% RSLogix 500 project LVD180611.RSS, saved by version 10.00.00.00 %
PROJECT "LINCEBOT"    % processor: MicroLogix 1400 %

PROGRAM FILES
  LAD 2 "MAIN"  15 rungs  % Main Program Routine %
  LAD 4 "PACKAGER"  10 rungs  % normal %
  LAD 6 "TIMING"  11 rungs  % normal %
  LAD 8 "LOOP TIME"  6 rungs
  LAD 10 "AIR PRESUR"  5 rungs
  LAD 12 "ENABLES"  10 rungs
  LAD 14 "SPEED OUT"  11 rungs
  LAD 70 "OFFSETS"  1 rungs  % normal %
  LAD 80 "HSC BOT"  9 rungs
  LAD 90 "HSC TOP"  9 rungs
  LAD 100 "1 MS STI"  23 rungs  % high speed %
  LAD 102 "SPEED BOT"  6 rungs  % high speed %
  LAD 103 "SPEED TOP"  6 rungs  % high speed %
  LAD 104 "P BOT"  8 rungs  % high speed %
  LAD 105 "P TOP"  8 rungs  % high speed %
  LAD 110 "SHIFT BOT"  5 rungs
  LAD 111 "SHIFT TOP"  5 rungs
  LAD 121 "OPTIC BOT"  23 rungs
  LAD 125 "INS 1"  61 rungs
  LAD 130 "XFER"  6 rungs
  LAD 140 "OPTIC TOP"  37 rungs
  LAD 150 "INS 5"  61 rungs
  LAD 160 "INS 6"  61 rungs
  LAD 170 "PASS BLOW"  3 rungs

DATA FILES
  O0 OUTPUT  11 elements
  I1 INPUT  11 elements
  S2 STATUS  66 elements
  B3 BINARY  14 elements
  T4 TIMER  40 elements
  C5 COUNTER  1 elements
  R6 CONTROL  10 elements
  N7 INTEGER  200 elements
  F8 FLOAT  100 elements
  B9 TOP BS DAT  256 elements
  B10 OLD_COM  1 elements
  B11 BOT BS DAT  256 elements
  B12 HMI_BINARY  22 elements  % general use with hmi to avoid additional reads %
  L13  COUNTS  100 elements
  F14 HMI_FLOAT  100 elements
  N15 HMI_INTS  100 elements
  L16 HMI_LONGS  100 elements
  L23 NEW READ  100 elements
  L24 NEW WRITE  100 elements
  L42   52 elements
  B181 BLANK  128 elements  % used to wipe bs files %
  F182 TEST FLOAT  50 elements
  L183 TEST LONG  50 elements
  N184 TEST INTS  50 elements
  B185 TEST BITS  50 elements
  N186 HMI INTS  50 elements
  L187 HMI LONG  50 elements
  F188 HMI FLOAT  50 elements
  B189 HMI BITS  50 elements
  L190 COUNTS  50 elements
  B191 ERROR BITS  10 elements
  L192 SPD OFFSET  50 elements
  F193 SPD OFFSET  50 elements
  B194 BOT GOOD  128 elements
  B195 TOP GOOD  128 elements
  B196 CTRL BITS  50 elements
  N197 CTRL INTS  50 elements
  B198 TRK BITS  50 elements
  L199 TRK LONG  50 elements
  N200 TRK INTS  50 elements
  L201 INS LONG  50 elements
  B202 INS BITS  50 elements
  N203 INS INTS  50 elements
  L204 CTRL LONG  50 elements
  F205 CTRL FLTS  50 elements

LADDER 2 "MAIN"    % Main Program Routine %
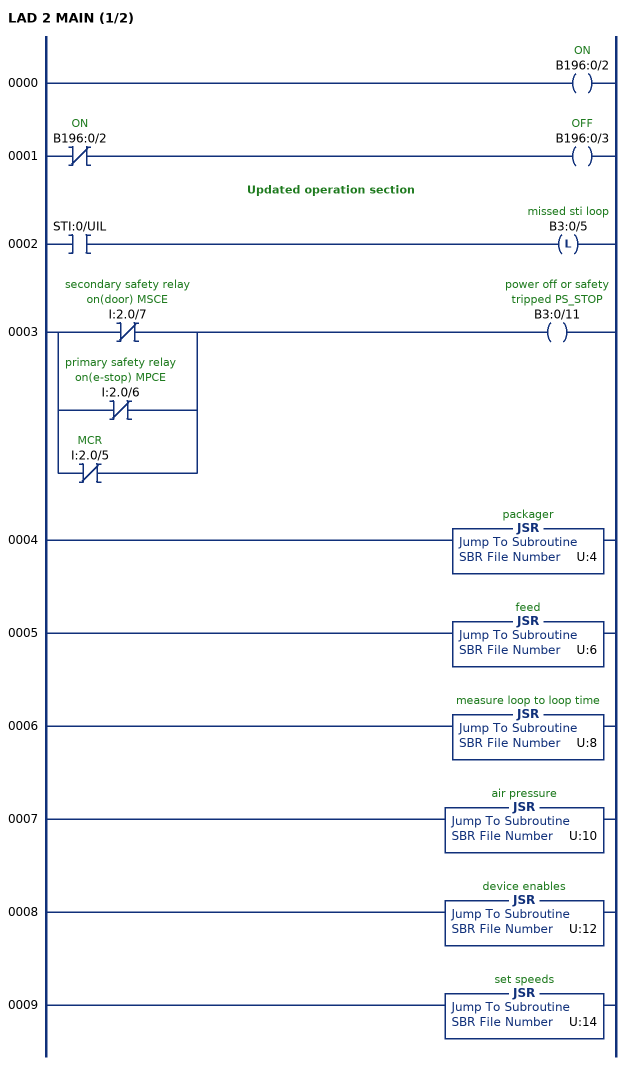
% Rung: 0 %
SOR OTE B196:0/2 EOR
%   B196:0/2  ON %
% Rung: 1 %
SOR XIO B196:0/2 OTE B196:0/3 EOR
%   B196:0/2  ON %
%   B196:0/3  OFF %
% Rung: 2 %
% TITLE: Updated operation section %
SOR XIC STI:0/UIL OTL B3:0/5 EOR
%   B3:0/5  "missed sti loop" %
% Rung: 3 %
SOR BST XIO I:2.0/7 NXB XIO I:2.0/6 NXB XIO I:2.0/5 BND OTE B3:0/11 EOR
%   I:2.0/7  MSCE  "secondary safety relay on(door)" %
%   I:2.0/6  MPCE  "primary safety relay on(e-stop)" %
%   I:2.0/5  MCR %
%   B3:0/11  PS_STOP  "power off or safety tripped" %
% Rung: 4 %
SOR JSR U:4 EOR
%   U:4  "packager" %
% Rung: 5 %
SOR JSR U:6 EOR
%   U:6  "feed" %
% Rung: 6 %
SOR JSR U:8 EOR
%   U:8  "measure loop to loop time" %
% Rung: 7 %
SOR JSR U:10 EOR
%   U:10  "air pressure" %
% Rung: 8 %
SOR JSR U:12 EOR
%   U:12  "device enables" %
% Rung: 9 %
SOR JSR U:14 EOR
%   U:14  "set speeds" %

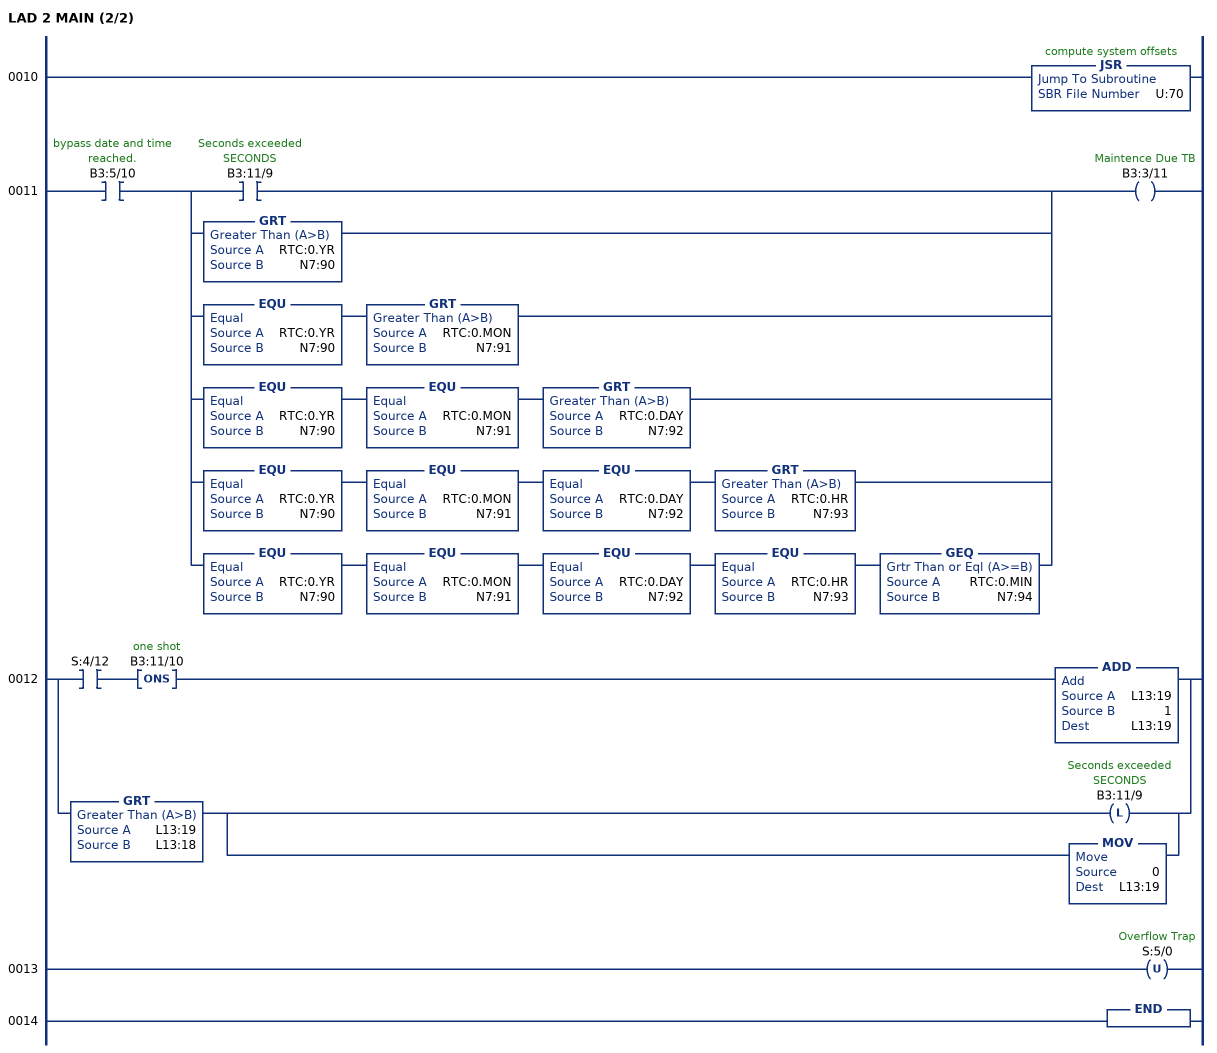
% Rung: 10 %
SOR JSR U:70 EOR
%   U:70  "compute system offsets" %
% Rung: 11 %
SOR XIC B3:5/10 BST XIC B3:11/9 NXB GRT RTC:0.YR N7:90 NXB EQU RTC:0.YR N7:90 GRT RTC:0.MON N7:91 NXB EQU RTC:0.YR N7:90 EQU RTC:0.MON N7:91 GRT RTC:0.DAY N7:92 NXB EQU RTC:0.YR N7:90 EQU RTC:0.MON N7:91 EQU RTC:0.DAY N7:92 GRT RTC:0.HR N7:93 NXB EQU RTC:0.YR N7:90 EQU RTC:0.MON N7:91 EQU RTC:0.DAY N7:92 EQU RTC:0.HR N7:93 GEQ RTC:0.MIN N7:94 BND OTE B3:3/11 EOR
%   B3:5/10  "bypass date and time reached." %
%   B3:11/9  SECONDS  "Seconds exceeded" %
%   N7:90  RTC %
%   B3:3/11  TB  "Maintence Due" %
% Rung: 12 %
SOR BST XIC S:4/12 ONS B3:11/10 ADD L13:19 1 L13:19 NXB GRT L13:19 L13:18 BST OTL B3:11/9 NXB MOV 0 L13:19 BND BND EOR
%   B3:11/10  "one shot" %
%   L13:18  MAX %
%   B3:11/9  SECONDS  "Seconds exceeded" %
% Rung: 13 %
SOR OTU S:5/0 EOR
%   S:5/0  "Overflow Trap" %
% Rung: 14 %
SOR END EOR

LADDER 4 "PACKAGER"    % normal %
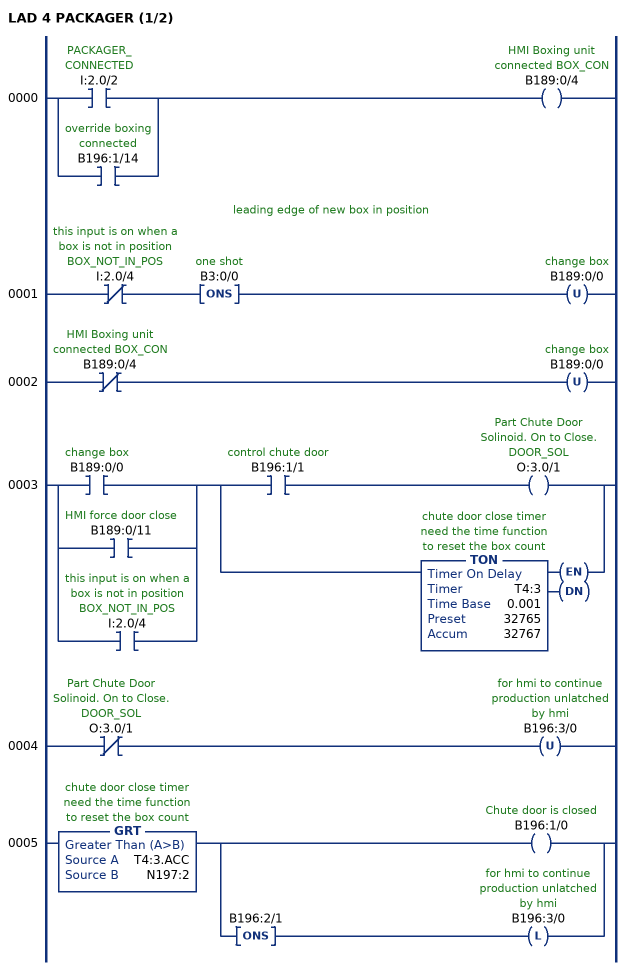
% Rung: 0 %
SOR BST XIC I:2.0/2 NXB XIC B196:1/14 BND OTE B189:0/4 EOR
%   I:2.0/2  PACKAGER_CONNECTED %
%   B196:1/14  "override boxing connected" %
%   B189:0/4  BOX_CON  "HMI Boxing unit connected" %
% Rung: 1 %
% leading edge of new box in position %
SOR XIO I:2.0/4 ONS B3:0/0 OTU B189:0/0 EOR
%   I:2.0/4  BOX_NOT_IN_POS  "this input is on when a box is not in position" %
%   B3:0/0  "one shot" %
%   B189:0/0  "change box" %
% Rung: 2 %
SOR XIO B189:0/4 OTU B189:0/0 EOR
%   B189:0/4  BOX_CON  "HMI Boxing unit connected" %
%   B189:0/0  "change box" %
% Rung: 3 %
SOR BST XIC B189:0/0 NXB XIC B189:0/11 NXB XIC I:2.0/4 BND BST XIC B196:1/1 OTE O:3.0/1 NXB TON T4:3 0.001 32765 32767 BND EOR
%   B189:0/0  "change box" %
%   B189:0/11  "HMI force door close" %
%   I:2.0/4  BOX_NOT_IN_POS  "this input is on when a box is not in position" %
%   B196:1/1  "control chute door" %
%   O:3.0/1  DOOR_SOL  "Part Chute Door Solinoid. On to Close." %
%   T4:3  "chute door close timer need the time function to reset the box count" %
% Rung: 4 %
SOR XIO O:3.0/1 OTU B196:3/0 EOR
%   O:3.0/1  DOOR_SOL  "Part Chute Door Solinoid. On to Close." %
%   B196:3/0  "for hmi to continue production unlatched by hmi" %
% Rung: 5 %
SOR GRT T4:3.ACC N197:2 BST OTE B196:1/0 NXB ONS B196:2/1 OTL B196:3/0 BND EOR
%   T4:3  "chute door close timer need the time function to reset the box count" %
%   N197:2  "time for chute door to close" %
%   B196:1/0  "Chute door is closed" %
%   B196:3/0  "for hmi to continue production unlatched by hmi" %

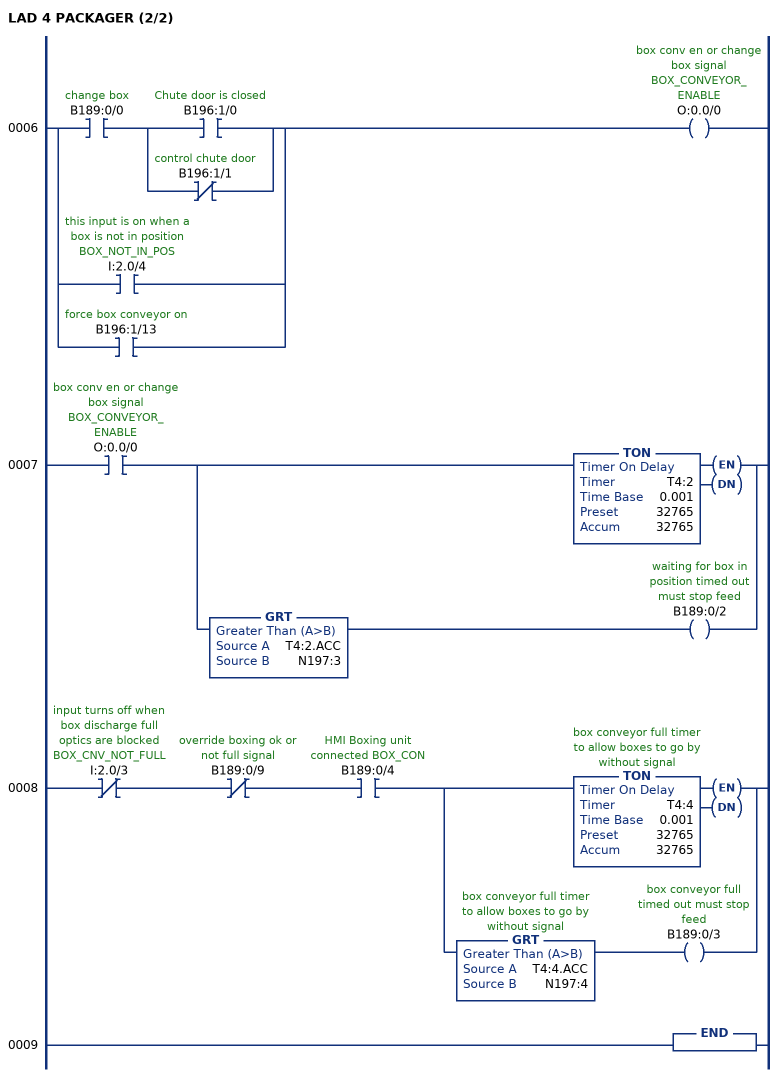
% Rung: 6 %
SOR BST XIC B189:0/0 BST XIC B196:1/0 NXB XIO B196:1/1 BND NXB XIC I:2.0/4 NXB XIC B196:1/13 BND OTE O:0.0/0 EOR
%   B189:0/0  "change box" %
%   B196:1/0  "Chute door is closed" %
%   B196:1/1  "control chute door" %
%   I:2.0/4  BOX_NOT_IN_POS  "this input is on when a box is not in position" %
%   B196:1/13  "force box conveyor on" %
%   O:0.0/0  BOX_CONVEYOR_ENABLE  "box conv en or change box signal" %
% Rung: 7 %
SOR XIC O:0.0/0 BST TON T4:2 0.001 32765 32765 NXB GRT T4:2.ACC N197:3 OTE B189:0/2 BND EOR
%   O:0.0/0  BOX_CONVEYOR_ENABLE  "box conv en or change box signal" %
%   N197:3  "FeedWheel Speed Output Setting" %
%   B189:0/2  "waiting for box in position timed out must stop feed" %
% Rung: 8 %
SOR XIO I:2.0/3 XIO B189:0/9 XIC B189:0/4 BST TON T4:4 0.001 32765 32765 NXB GRT T4:4.ACC N197:4 OTE B189:0/3 BND EOR
%   I:2.0/3  BOX_CNV_NOT_FULL  "input turns off when box discharge full optics are blocked" %
%   B189:0/9  "override boxing ok or not full signal" %
%   B189:0/4  BOX_CON  "HMI Boxing unit connected" %
%   T4:4  "box conveyor full timer to allow boxes to go by without signal" %
%   N197:4  "boxing convery full time out time (ms)" %
%   B189:0/3  "box conveyor full timed out must stop feed" %
% Rung: 9 %
SOR END EOR

LADDER 6 "TIMING"    % normal %
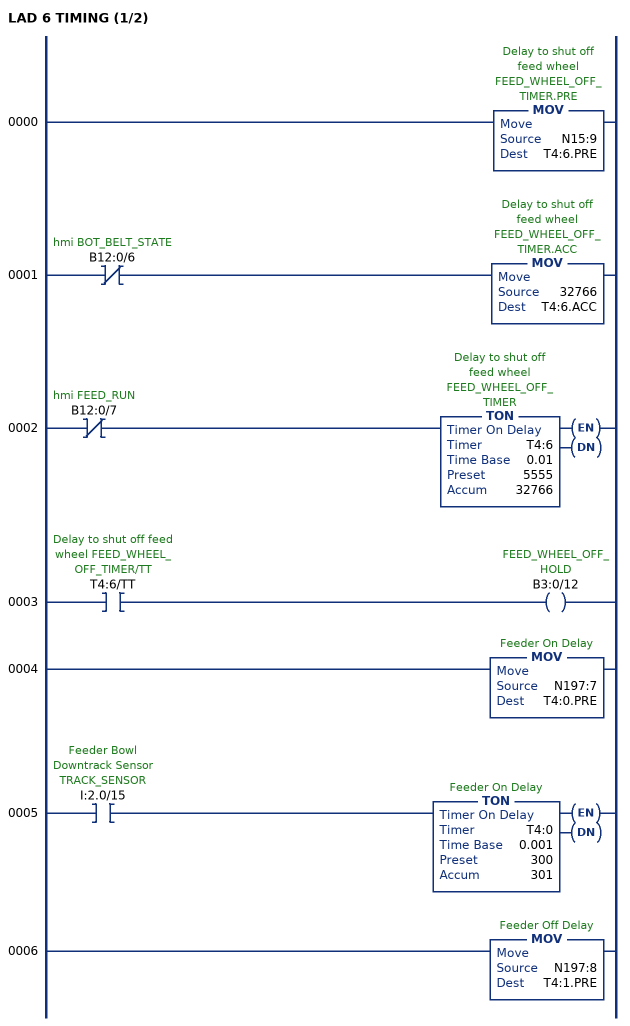
% Rung: 0 %
SOR MOV N15:9 T4:6.PRE EOR
%   N15:9  FEED_WHEEL_STOP_TIME %
%   T4:6  FEED_WHEEL_OFF_TIMER  "Delay to shut off feed wheel" %
% Rung: 1 %
SOR XIO B12:0/6 MOV 32766 T4:6.ACC EOR
%   B12:0/6  BOT_BELT_STATE  "hmi" %
%   T4:6  FEED_WHEEL_OFF_TIMER  "Delay to shut off feed wheel" %
% Rung: 2 %
SOR XIO B12:0/7 TON T4:6 0.01 5555 32766 EOR
%   B12:0/7  FEED_RUN  "hmi" %
%   T4:6  FEED_WHEEL_OFF_TIMER  "Delay to shut off feed wheel" %
% Rung: 3 %
SOR XIC T4:6/TT OTE B3:0/12 EOR
%   T4:6  FEED_WHEEL_OFF_TIMER  "Delay to shut off feed wheel" %
%   B3:0/12  FEED_WHEEL_OFF_HOLD %
% Rung: 4 %
SOR MOV N197:7 T4:0.PRE EOR
%   N197:7  "down track on delay" %
%   T4:0  "Feeder On Delay" %
% Rung: 5 %
SOR XIC I:2.0/15 TON T4:0 0.001 300 301 EOR
%   I:2.0/15  TRACK_SENSOR  "Feeder Bowl Downtrack Sensor" %
%   T4:0  "Feeder On Delay" %
% Rung: 6 %
SOR MOV N197:8 T4:1.PRE EOR
%   N197:8  "down track off delay" %
%   T4:1  "Feeder Off Delay" %

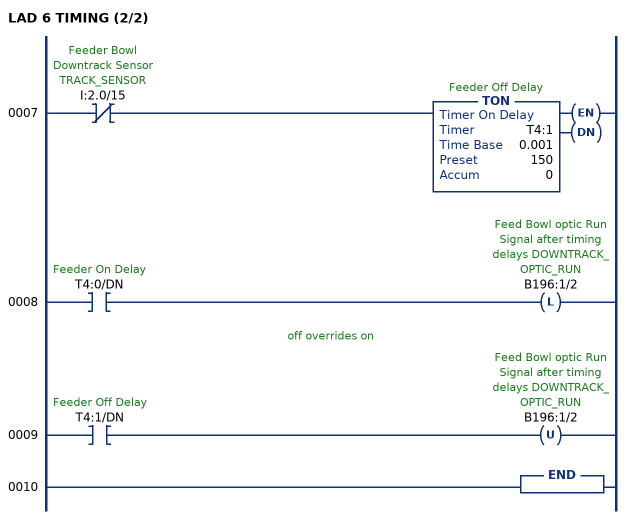
% Rung: 7 %
SOR XIO I:2.0/15 TON T4:1 0.001 150 0 EOR
%   I:2.0/15  TRACK_SENSOR  "Feeder Bowl Downtrack Sensor" %
%   T4:1  "Feeder Off Delay" %
% Rung: 8 %
SOR XIC T4:0/DN OTL B196:1/2 EOR
%   T4:0  "Feeder On Delay" %
%   B196:1/2  DOWNTRACK_OPTIC_RUN  "Feed Bowl optic Run Signal after timing delays" %
% Rung: 9 %
% off overrides on %
SOR XIC T4:1/DN OTU B196:1/2 EOR
%   T4:1  "Feeder Off Delay" %
%   B196:1/2  DOWNTRACK_OPTIC_RUN  "Feed Bowl optic Run Signal after timing delays" %
% Rung: 10 %
SOR END EOR

LADDER 8 "LOOP TIME"
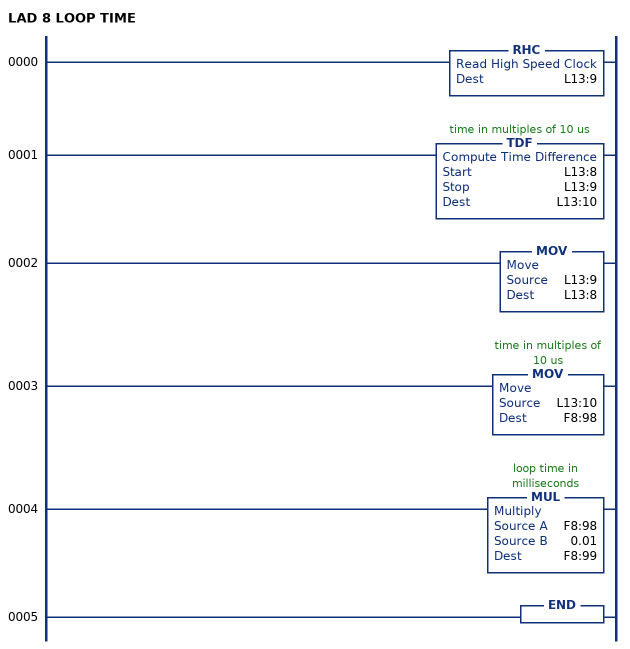
% Rung: 0 %
SOR RHC L13:9 EOR
% Rung: 1 %
SOR TDF L13:8 L13:9 L13:10 EOR
%   L13:10  "time in multiples of 10 us" %
% Rung: 2 %
SOR MOV L13:9 L13:8 EOR
% Rung: 3 %
SOR MOV L13:10 F8:98 EOR
%   L13:10  "time in multiples of 10 us" %
%   F8:98  "time in multiples of 10 us" %
% Rung: 4 %
SOR MUL F8:98 0.01 F8:99 EOR
%   F8:98  "time in multiples of 10 us" %
%   F8:99  "loop time in milliseconds" %
% Rung: 5 %
SOR END EOR

LADDER 10 "AIR PRESUR"
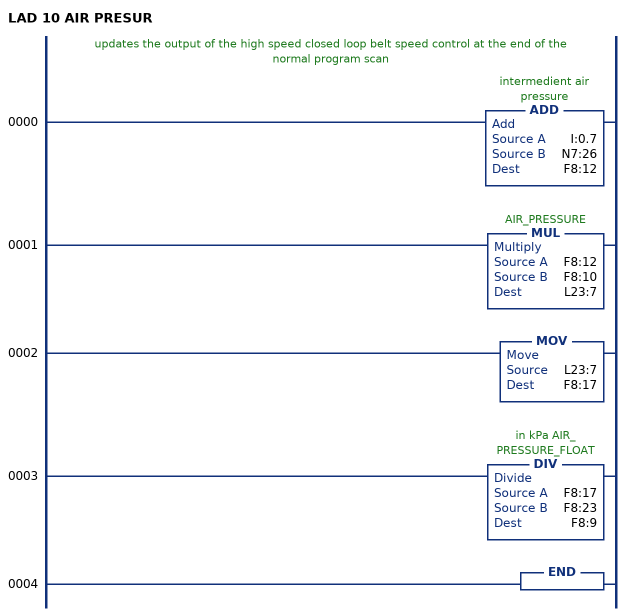
% Rung: 0 %
% updates the output of the high speed closed loop belt speed control at the end of the normal program scan %
SOR ADD I:0.7 N7:26 F8:12 EOR
%   I:0.7  "Air Presure Sensor Input Signal" %
%   N7:26  MAIN_AIR_OFFSET  "Main Air Offset old machine -398 new machine 0" %
%   F8:12  "intermedient air pressure" %
% Rung: 1 %
SOR MUL F8:12 F8:10 L23:7 EOR
%   F8:12  "intermedient air pressure" %
%   F8:10  AIR_MULTIPLIER_BAR  "Air Multiplier (BAR)" %
%   L23:7  AIR_PRESSURE %
% Rung: 2 %
SOR MOV L23:7 F8:17 EOR
%   L23:7  AIR_PRESSURE %
% Rung: 3 %
SOR DIV F8:17 F8:23 F8:9 EOR
%   F8:9  AIR_PRESSURE_FLOAT  "in kPa" %
% Rung: 4 %
SOR END EOR

LADDER 12 "ENABLES"
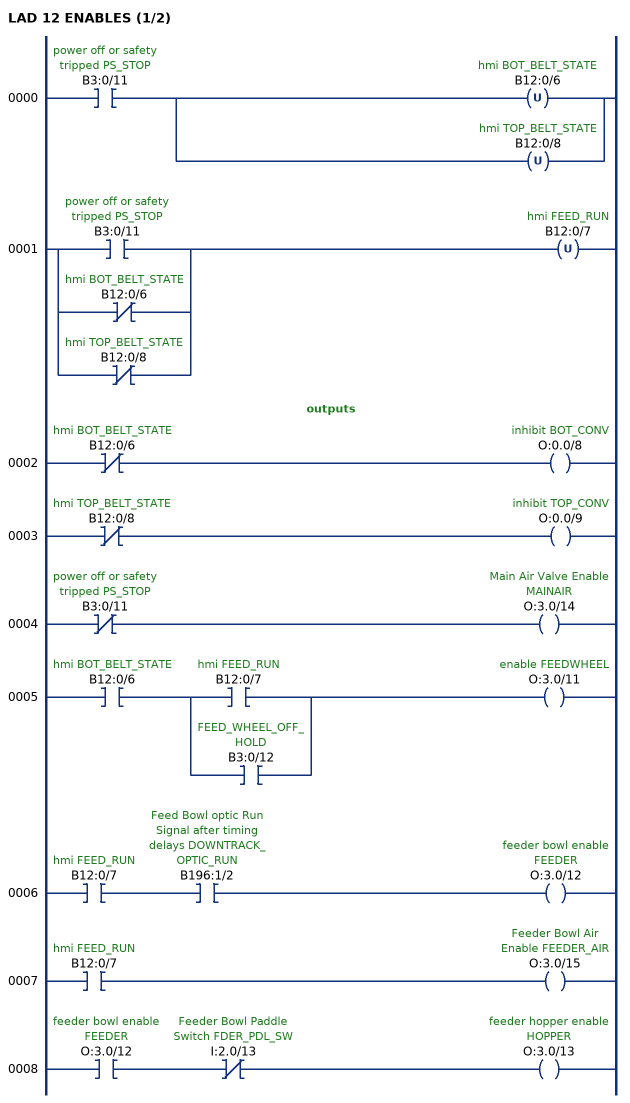
% Rung: 0 %
SOR XIC B3:0/11 BST OTU B12:0/6 NXB OTU B12:0/8 BND EOR
%   B3:0/11  PS_STOP  "power off or safety tripped" %
%   B12:0/6  BOT_BELT_STATE  "hmi" %
%   B12:0/8  TOP_BELT_STATE  "hmi" %
% Rung: 1 %
SOR BST XIC B3:0/11 NXB XIO B12:0/6 NXB XIO B12:0/8 BND OTU B12:0/7 EOR
%   B3:0/11  PS_STOP  "power off or safety tripped" %
%   B12:0/6  BOT_BELT_STATE  "hmi" %
%   B12:0/8  TOP_BELT_STATE  "hmi" %
%   B12:0/7  FEED_RUN  "hmi" %
% Rung: 2 %
% TITLE: outputs %
SOR XIO B12:0/6 OTE O:0.0/8 EOR
%   B12:0/6  BOT_BELT_STATE  "hmi" %
%   O:0.0/8  BOT_CONV  "inhibit" %
% Rung: 3 %
SOR XIO B12:0/8 OTE O:0.0/9 EOR
%   B12:0/8  TOP_BELT_STATE  "hmi" %
%   O:0.0/9  TOP_CONV  "inhibit" %
% Rung: 4 %
SOR XIO B3:0/11 OTE O:3.0/14 EOR
%   B3:0/11  PS_STOP  "power off or safety tripped" %
%   O:3.0/14  MAINAIR  "Main Air Valve Enable" %
% Rung: 5 %
SOR XIC B12:0/6 BST XIC B12:0/7 NXB XIC B3:0/12 BND OTE O:3.0/11 EOR
%   B12:0/6  BOT_BELT_STATE  "hmi" %
%   B12:0/7  FEED_RUN  "hmi" %
%   B3:0/12  FEED_WHEEL_OFF_HOLD %
%   O:3.0/11  FEEDWHEEL  "enable" %
% Rung: 6 %
SOR XIC B12:0/7 XIC B196:1/2 OTE O:3.0/12 EOR
%   B12:0/7  FEED_RUN  "hmi" %
%   B196:1/2  DOWNTRACK_OPTIC_RUN  "Feed Bowl optic Run Signal after timing delays" %
%   O:3.0/12  FEEDER  "feeder bowl enable" %
% Rung: 7 %
SOR XIC B12:0/7 OTE O:3.0/15 EOR
%   B12:0/7  FEED_RUN  "hmi" %
%   O:3.0/15  FEEDER_AIR  "Feeder Bowl Air Enable" %
% Rung: 8 %
SOR XIC O:3.0/12 XIO I:2.0/13 OTE O:3.0/13 EOR
%   O:3.0/12  FEEDER  "feeder bowl enable" %
%   I:2.0/13  FDER_PDL_SW  "Feeder Bowl Paddle Switch" %
%   O:3.0/13  HOPPER  "feeder hopper enable" %

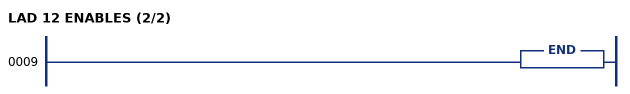
% Rung: 9 %
SOR END EOR

LADDER 14 "SPEED OUT"
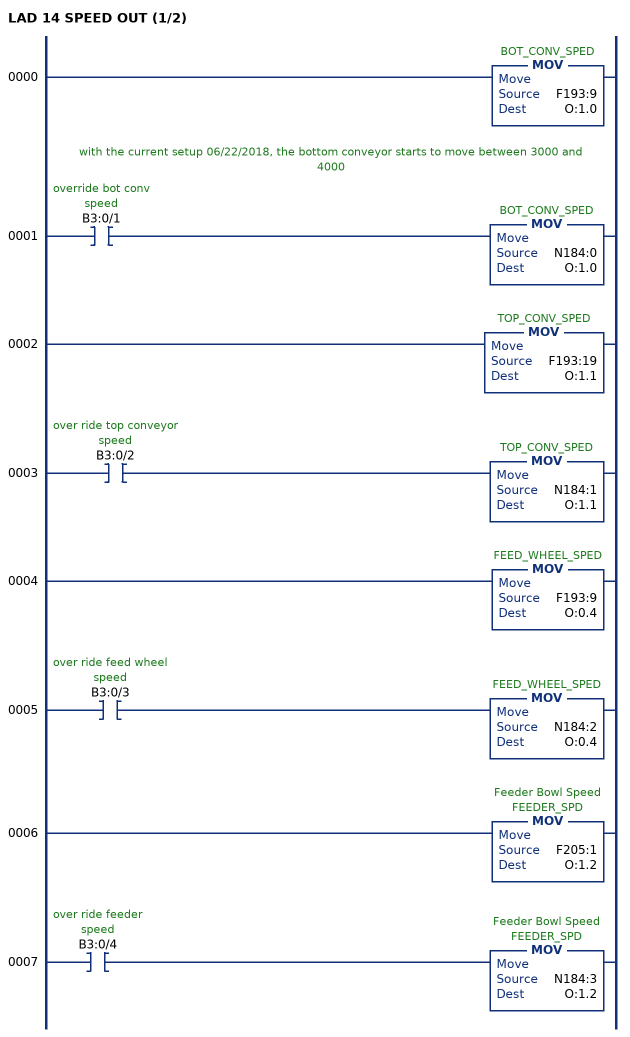
% Rung: 0 %
SOR MOV F193:9 O:1.0 EOR
%   F193:9  SCALED_BOT_VALUE %
%   O:1.0  BOT_CONV_SPED %
% Rung: 1 %
% with the current setup 06/22/2018, the bottom conveyor starts to move between 3000 and 4000 %
SOR XIC B3:0/1 MOV N184:0 O:1.0 EOR
%   B3:0/1  "override bot conv speed" %
%   O:1.0  BOT_CONV_SPED %
% Rung: 2 %
SOR MOV F193:19 O:1.1 EOR
%   F193:19  SCALED_TOP_VALUE %
%   O:1.1  TOP_CONV_SPED %
% Rung: 3 %
SOR XIC B3:0/2 MOV N184:1 O:1.1 EOR
%   B3:0/2  "over ride top conveyor speed" %
%   O:1.1  TOP_CONV_SPED %
% Rung: 4 %
SOR MOV F193:9 O:0.4 EOR
%   F193:9  SCALED_BOT_VALUE %
%   O:0.4  FEED_WHEEL_SPED %
% Rung: 5 %
SOR XIC B3:0/3 MOV N184:2 O:0.4 EOR
%   B3:0/3  "over ride feed wheel speed" %
%   O:0.4  FEED_WHEEL_SPED %
% Rung: 6 %
SOR MOV F205:1 O:1.2 EOR
%   F205:1  "feed bowl" %
%   O:1.2  FEEDER_SPD  "Feeder Bowl Speed" %
% Rung: 7 %
SOR XIC B3:0/4 MOV N184:3 O:1.2 EOR
%   B3:0/4  "over ride feeder speed" %
%   O:1.2  FEEDER_SPD  "Feeder Bowl Speed" %

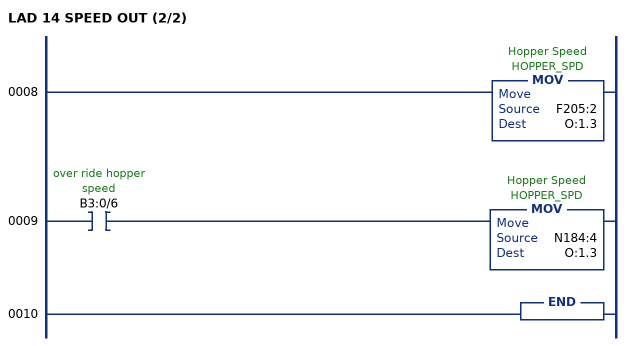
% Rung: 8 %
SOR MOV F205:2 O:1.3 EOR
%   F205:2  "hopper" %
%   O:1.3  HOPPER_SPD  "Hopper Speed" %
% Rung: 9 %
SOR XIC B3:0/6 MOV N184:4 O:1.3 EOR
%   B3:0/6  "over ride hopper speed" %
%   O:1.3  HOPPER_SPD  "Hopper Speed" %
% Rung: 10 %
SOR END EOR

LADDER 80 "HSC BOT"
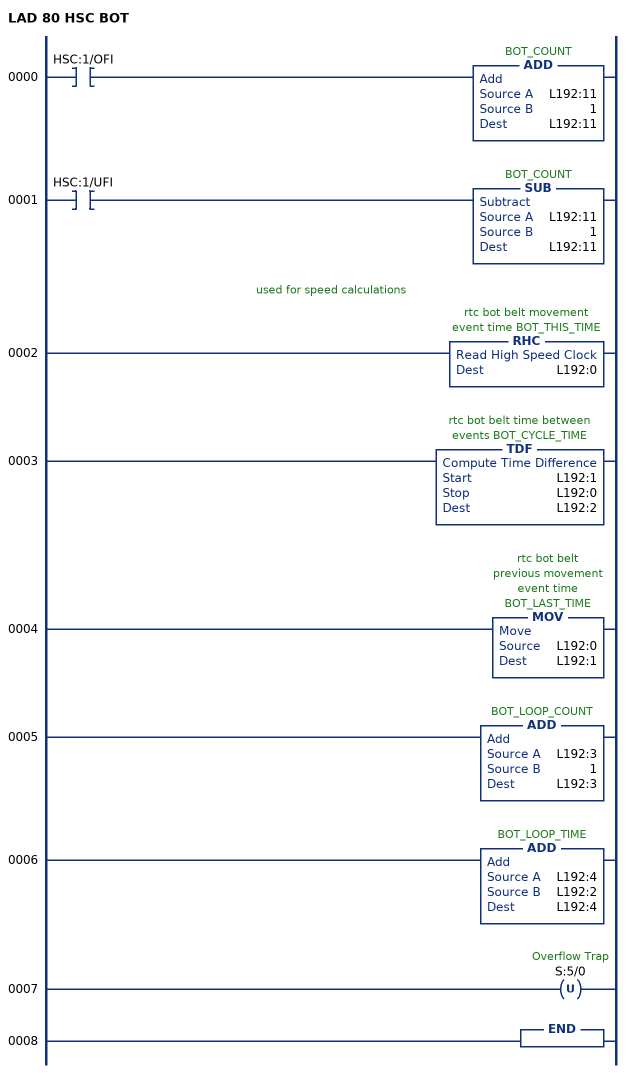
% Rung: 0 %
SOR XIC HSC:1/OFI ADD L192:11 1 L192:11 EOR
%   L192:11  BOT_COUNT %
% Rung: 1 %
SOR XIC HSC:1/UFI SUB L192:11 1 L192:11 EOR
%   L192:11  BOT_COUNT %
% Rung: 2 %
% used for speed calculations %
SOR RHC L192:0 EOR
%   L192:0  BOT_THIS_TIME  "rtc bot belt movement event time" %
% Rung: 3 %
SOR TDF L192:1 L192:0 L192:2 EOR
%   L192:1  BOT_LAST_TIME  "rtc bot belt previous movement event time" %
%   L192:0  BOT_THIS_TIME  "rtc bot belt movement event time" %
%   L192:2  BOT_CYCLE_TIME  "rtc bot belt time between events" %
% Rung: 4 %
SOR MOV L192:0 L192:1 EOR
%   L192:0  BOT_THIS_TIME  "rtc bot belt movement event time" %
%   L192:1  BOT_LAST_TIME  "rtc bot belt previous movement event time" %
% Rung: 5 %
SOR ADD L192:3 1 L192:3 EOR
%   L192:3  BOT_LOOP_COUNT %
% Rung: 6 %
SOR ADD L192:4 L192:2 L192:4 EOR
%   L192:4  BOT_LOOP_TIME %
%   L192:2  BOT_CYCLE_TIME  "rtc bot belt time between events" %
% Rung: 7 %
SOR OTU S:5/0 EOR
%   S:5/0  "Overflow Trap" %
% Rung: 8 %
SOR END EOR

LADDER 90 "HSC TOP"
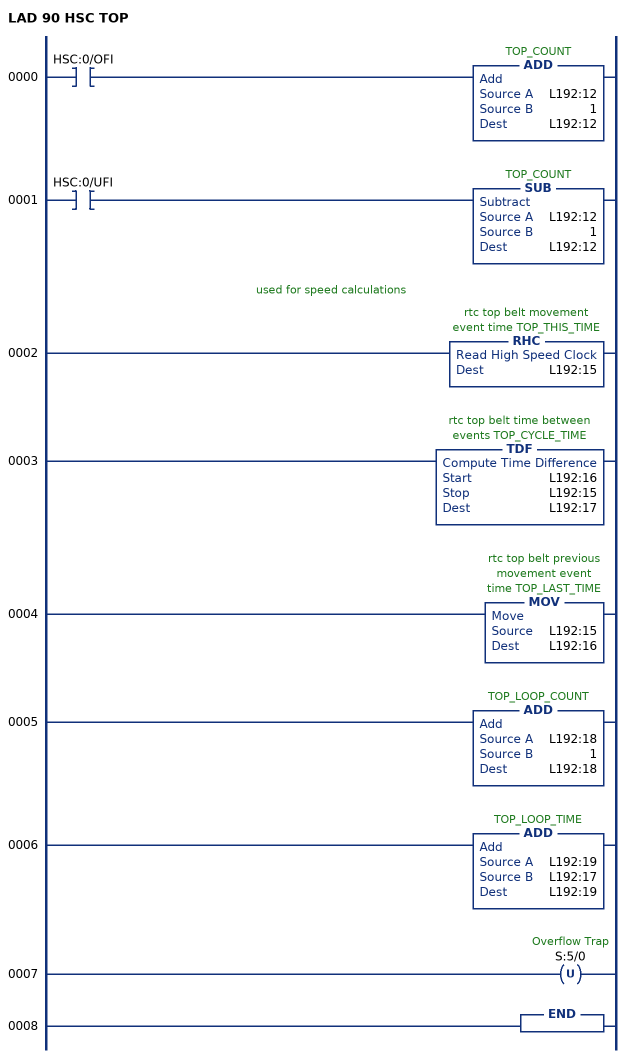
% Rung: 0 %
SOR XIC HSC:0/OFI ADD L192:12 1 L192:12 EOR
%   L192:12  TOP_COUNT %
% Rung: 1 %
SOR XIC HSC:0/UFI SUB L192:12 1 L192:12 EOR
%   L192:12  TOP_COUNT %
% Rung: 2 %
% used for speed calculations %
SOR RHC L192:15 EOR
%   L192:15  TOP_THIS_TIME  "rtc top belt movement event time" %
% Rung: 3 %
SOR TDF L192:16 L192:15 L192:17 EOR
%   L192:16  TOP_LAST_TIME  "rtc top belt previous movement event time" %
%   L192:15  TOP_THIS_TIME  "rtc top belt movement event time" %
%   L192:17  TOP_CYCLE_TIME  "rtc top belt time between events" %
% Rung: 4 %
SOR MOV L192:15 L192:16 EOR
%   L192:15  TOP_THIS_TIME  "rtc top belt movement event time" %
%   L192:16  TOP_LAST_TIME  "rtc top belt previous movement event time" %
% Rung: 5 %
SOR ADD L192:18 1 L192:18 EOR
%   L192:18  TOP_LOOP_COUNT %
% Rung: 6 %
SOR ADD L192:19 L192:17 L192:19 EOR
%   L192:19  TOP_LOOP_TIME %
%   L192:17  TOP_CYCLE_TIME  "rtc top belt time between events" %
% Rung: 7 %
SOR OTU S:5/0 EOR
%   S:5/0  "Overflow Trap" %
% Rung: 8 %
SOR END EOR

LADDER 100 "1 MS STI"    % high speed %
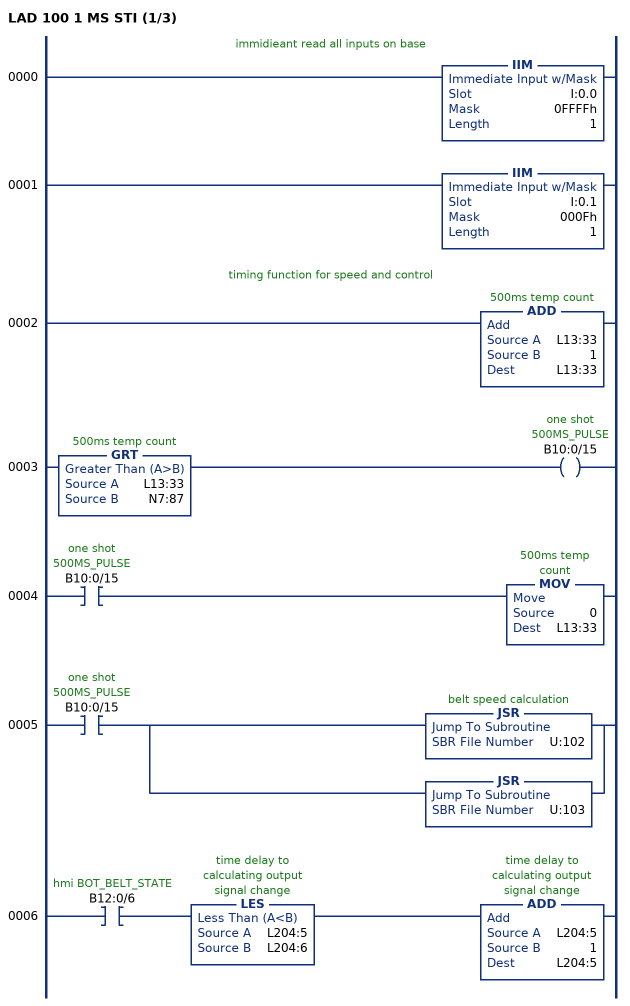
% Rung: 0 %
% immidieant read all inputs on base %
SOR IIM I:0.0 0FFFFh 1 EOR
% Rung: 1 %
SOR IIM I:0.1 000Fh 1 EOR
% Rung: 2 %
% timing function for speed and control %
SOR ADD L13:33 1 L13:33 EOR
%   L13:33  "500ms temp count" %
% Rung: 3 %
SOR GRT L13:33 N7:87 OTE B10:0/15 EOR
%   L13:33  "500ms temp count" %
%   B10:0/15  500MS_PULSE  "one shot" %
% Rung: 4 %
SOR XIC B10:0/15 MOV 0 L13:33 EOR
%   B10:0/15  500MS_PULSE  "one shot" %
%   L13:33  "500ms temp count" %
% Rung: 5 %
SOR XIC B10:0/15 BST JSR U:102 NXB JSR U:103 BND EOR
%   B10:0/15  500MS_PULSE  "one shot" %
%   U:102  "belt speed calculation" %
% Rung: 6 %
SOR XIC B12:0/6 LES L204:5 L204:6 ADD L204:5 1 L204:5 EOR
%   B12:0/6  BOT_BELT_STATE  "hmi" %
%   L204:5  "time delay to calculating output signal change" %
%   L204:6  "belt start delay time" %

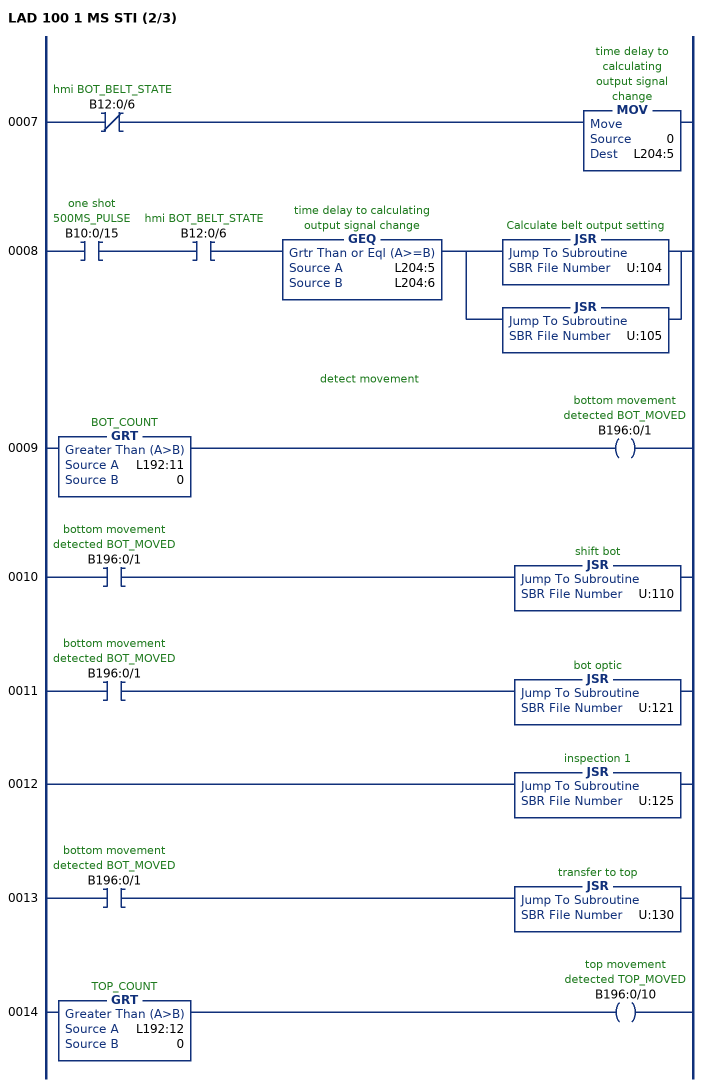
% Rung: 7 %
SOR XIO B12:0/6 MOV 0 L204:5 EOR
%   B12:0/6  BOT_BELT_STATE  "hmi" %
%   L204:5  "time delay to calculating output signal change" %
% Rung: 8 %
SOR XIC B10:0/15 XIC B12:0/6 GEQ L204:5 L204:6 BST JSR U:104 NXB JSR U:105 BND EOR
%   B10:0/15  500MS_PULSE  "one shot" %
%   B12:0/6  BOT_BELT_STATE  "hmi" %
%   L204:5  "time delay to calculating output signal change" %
%   L204:6  "belt start delay time" %
%   U:104  "Calculate belt output setting" %
% Rung: 9 %
% detect movement %
SOR GRT L192:11 0 OTE B196:0/1 EOR
%   L192:11  BOT_COUNT %
%   B196:0/1  BOT_MOVED  "bottom movement detected" %
% Rung: 10 %
SOR XIC B196:0/1 JSR U:110 EOR
%   B196:0/1  BOT_MOVED  "bottom movement detected" %
%   U:110  "shift bot" %
% Rung: 11 %
SOR XIC B196:0/1 JSR U:121 EOR
%   B196:0/1  BOT_MOVED  "bottom movement detected" %
%   U:121  "bot optic" %
% Rung: 12 %
SOR JSR U:125 EOR
%   U:125  "inspection 1" %
% Rung: 13 %
SOR XIC B196:0/1 JSR U:130 EOR
%   B196:0/1  BOT_MOVED  "bottom movement detected" %
%   U:130  "transfer to top" %
% Rung: 14 %
SOR GRT L192:12 0 OTE B196:0/10 EOR
%   L192:12  TOP_COUNT %
%   B196:0/10  TOP_MOVED  "top movement detected" %

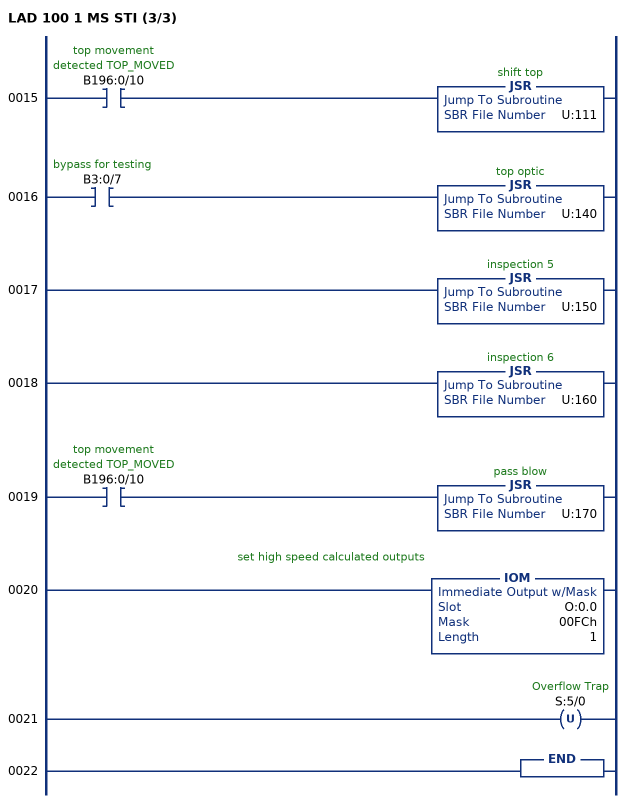
% Rung: 15 %
SOR XIC B196:0/10 JSR U:111 EOR
%   B196:0/10  TOP_MOVED  "top movement detected" %
%   U:111  "shift top" %
% Rung: 16 %
SOR XIC B3:0/7 JSR U:140 EOR
%   B3:0/7  "bypass for testing" %
%   U:140  "top optic" %
% Rung: 17 %
SOR JSR U:150 EOR
%   U:150  "inspection 5" %
% Rung: 18 %
SOR JSR U:160 EOR
%   U:160  "inspection 6" %
% Rung: 19 %
SOR XIC B196:0/10 JSR U:170 EOR
%   B196:0/10  TOP_MOVED  "top movement detected" %
%   U:170  "pass blow" %
% Rung: 20 %
% set high speed calculated outputs %
SOR IOM O:0.0 00FCh 1 EOR
% Rung: 21 %
SOR OTU S:5/0 EOR
%   S:5/0  "Overflow Trap" %
% Rung: 22 %
SOR END EOR

LADDER 102 "SPEED BOT"    % high speed %
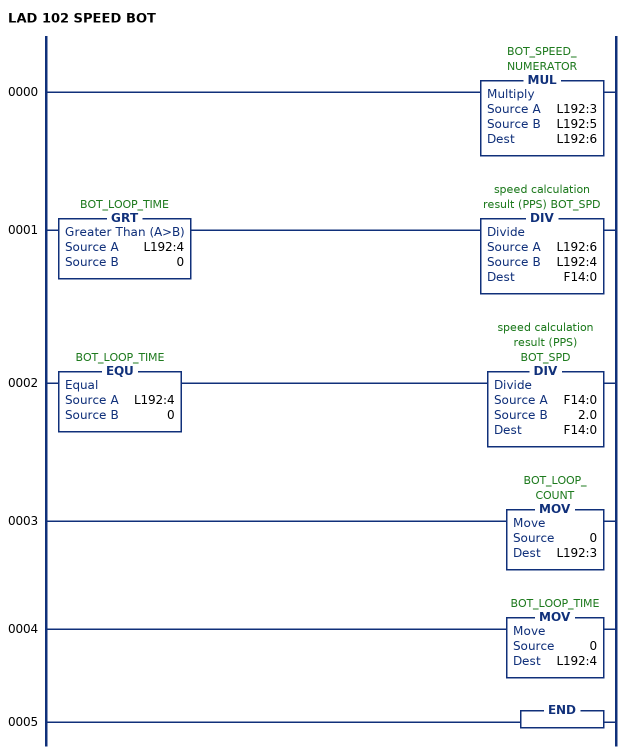
% Rung: 0 %
SOR MUL L192:3 L192:5 L192:6 EOR
%   L192:3  BOT_LOOP_COUNT %
%   L192:5  TKS_PER_SECOND %
%   L192:6  BOT_SPEED_NUMERATOR %
% Rung: 1 %
SOR GRT L192:4 0 DIV L192:6 L192:4 F14:0 EOR
%   L192:4  BOT_LOOP_TIME %
%   L192:6  BOT_SPEED_NUMERATOR %
%   F14:0  BOT_SPD  "speed calculation result (PPS)" %
% Rung: 2 %
SOR EQU L192:4 0 DIV F14:0 2.0 F14:0 EOR
%   L192:4  BOT_LOOP_TIME %
%   F14:0  BOT_SPD  "speed calculation result (PPS)" %
% Rung: 3 %
SOR MOV 0 L192:3 EOR
%   L192:3  BOT_LOOP_COUNT %
% Rung: 4 %
SOR MOV 0 L192:4 EOR
%   L192:4  BOT_LOOP_TIME %
% Rung: 5 %
SOR END EOR

LADDER 103 "SPEED TOP"    % high speed %
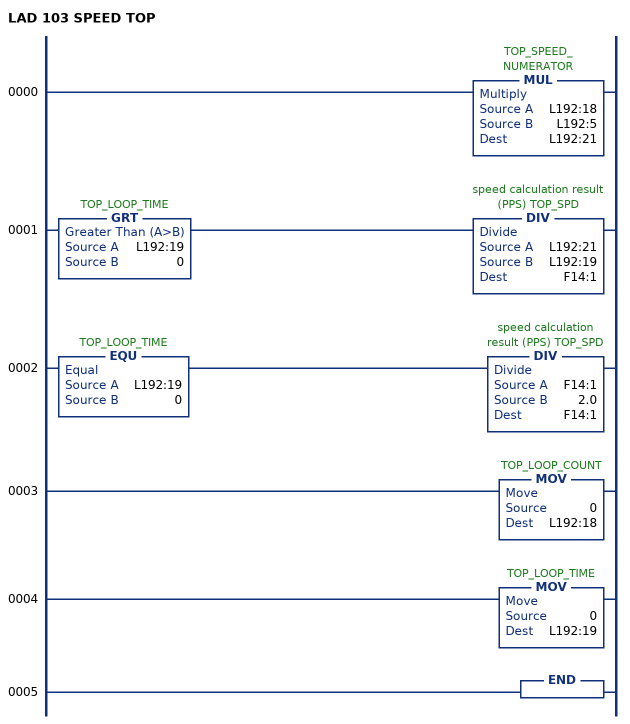
% Rung: 0 %
SOR MUL L192:18 L192:5 L192:21 EOR
%   L192:18  TOP_LOOP_COUNT %
%   L192:5  TKS_PER_SECOND %
%   L192:21  TOP_SPEED_NUMERATOR %
% Rung: 1 %
SOR GRT L192:19 0 DIV L192:21 L192:19 F14:1 EOR
%   L192:19  TOP_LOOP_TIME %
%   L192:21  TOP_SPEED_NUMERATOR %
%   F14:1  TOP_SPD  "speed calculation result (PPS)" %
% Rung: 2 %
SOR EQU L192:19 0 DIV F14:1 2.0 F14:1 EOR
%   L192:19  TOP_LOOP_TIME %
%   F14:1  TOP_SPD  "speed calculation result (PPS)" %
% Rung: 3 %
SOR MOV 0 L192:18 EOR
%   L192:18  TOP_LOOP_COUNT %
% Rung: 4 %
SOR MOV 0 L192:19 EOR
%   L192:19  TOP_LOOP_TIME %
% Rung: 5 %
SOR END EOR

LADDER 104 "P BOT"    % high speed %
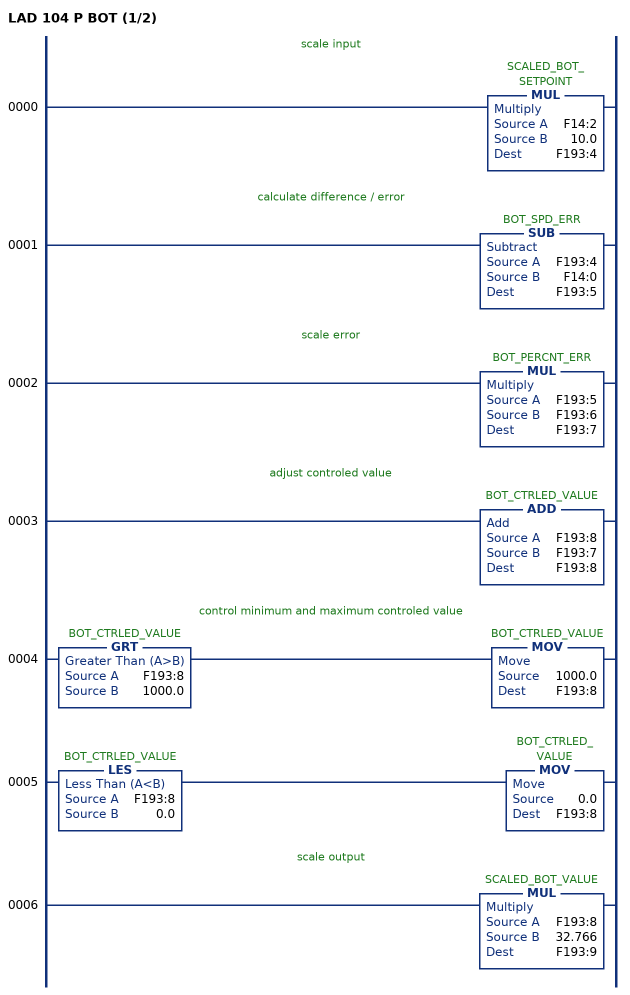
% Rung: 0 %
% scale input %
SOR MUL F14:2 10.0 F193:4 EOR
%   F14:2  BOT_SPD_SETPOINT %
%   F193:4  SCALED_BOT_SETPOINT %
% Rung: 1 %
% calculate difference / error %
SOR SUB F193:4 F14:0 F193:5 EOR
%   F193:4  SCALED_BOT_SETPOINT %
%   F14:0  BOT_SPD  "speed calculation result (PPS)" %
%   F193:5  BOT_SPD_ERR %
% Rung: 2 %
% scale error %
SOR MUL F193:5 F193:6 F193:7 EOR
%   F193:5  BOT_SPD_ERR %
%   F193:6  BOT_FDBK_RATIO %
%   F193:7  BOT_PERCNT_ERR %
% Rung: 3 %
% adjust controled value %
SOR ADD F193:8 F193:7 F193:8 EOR
%   F193:8  BOT_CTRLED_VALUE %
%   F193:7  BOT_PERCNT_ERR %
% Rung: 4 %
% control minimum and maximum controled value %
SOR GRT F193:8 1000.0 MOV 1000.0 F193:8 EOR
%   F193:8  BOT_CTRLED_VALUE %
% Rung: 5 %
SOR LES F193:8 0.0 MOV 0.0 F193:8 EOR
%   F193:8  BOT_CTRLED_VALUE %
% Rung: 6 %
% scale output %
SOR MUL F193:8 32.766 F193:9 EOR
%   F193:8  BOT_CTRLED_VALUE %
%   F193:9  SCALED_BOT_VALUE %

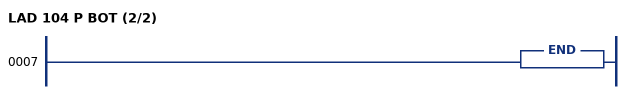
% Rung: 7 %
SOR END EOR

LADDER 105 "P TOP"    % high speed %
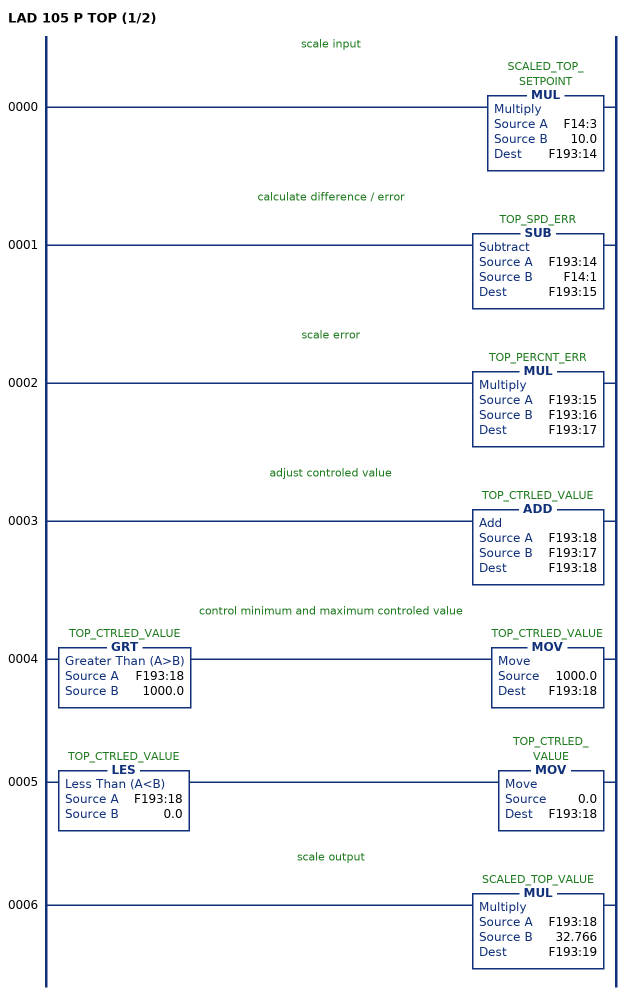
% Rung: 0 %
% scale input %
SOR MUL F14:3 10.0 F193:14 EOR
%   F14:3  TOP_SPD_SETPOINT %
%   F193:14  SCALED_TOP_SETPOINT %
% Rung: 1 %
% calculate difference / error %
SOR SUB F193:14 F14:1 F193:15 EOR
%   F193:14  SCALED_TOP_SETPOINT %
%   F14:1  TOP_SPD  "speed calculation result (PPS)" %
%   F193:15  TOP_SPD_ERR %
% Rung: 2 %
% scale error %
SOR MUL F193:15 F193:16 F193:17 EOR
%   F193:15  TOP_SPD_ERR %
%   F193:16  TOP_FDBK_RATIO %
%   F193:17  TOP_PERCNT_ERR %
% Rung: 3 %
% adjust controled value %
SOR ADD F193:18 F193:17 F193:18 EOR
%   F193:18  TOP_CTRLED_VALUE %
%   F193:17  TOP_PERCNT_ERR %
% Rung: 4 %
% control minimum and maximum controled value %
SOR GRT F193:18 1000.0 MOV 1000.0 F193:18 EOR
%   F193:18  TOP_CTRLED_VALUE %
% Rung: 5 %
SOR LES F193:18 0.0 MOV 0.0 F193:18 EOR
%   F193:18  TOP_CTRLED_VALUE %
% Rung: 6 %
% scale output %
SOR MUL F193:18 32.766 F193:19 EOR
%   F193:18  TOP_CTRLED_VALUE %
%   F193:19  SCALED_TOP_VALUE %

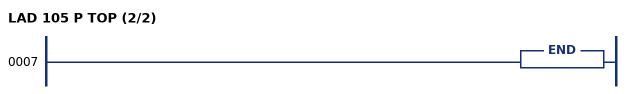
% Rung: 7 %
SOR END EOR

LADDER 110 "SHIFT BOT"
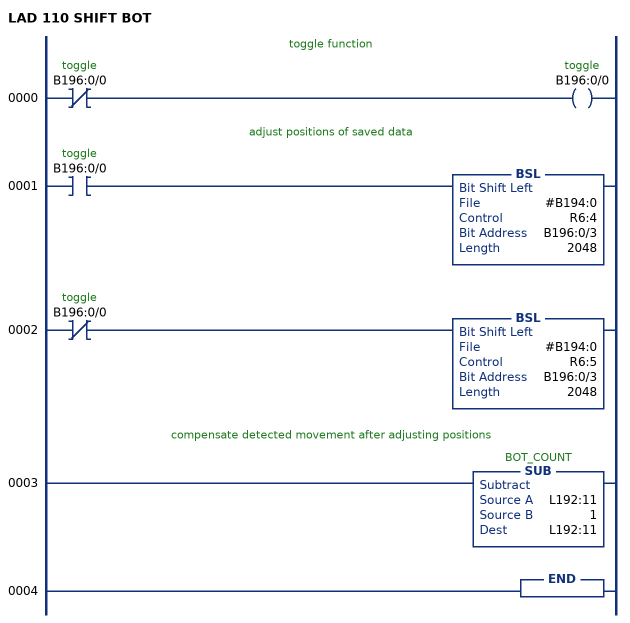
% Rung: 0 %
% toggle function %
SOR XIO B196:0/0 OTE B196:0/0 EOR
%   B196:0/0  "toggle" %
% Rung: 1 %
% adjust positions of saved data %
SOR XIC B196:0/0 BSL #B194:0 R6:4 B196:0/3 2048 EOR
%   B196:0/0  "toggle" %
%   B196:0/3  OFF %
% Rung: 2 %
SOR XIO B196:0/0 BSL #B194:0 R6:5 B196:0/3 2048 EOR
%   B196:0/0  "toggle" %
%   B196:0/3  OFF %
% Rung: 3 %
% compensate detected movement after adjusting positions %
SOR SUB L192:11 1 L192:11 EOR
%   L192:11  BOT_COUNT %
% Rung: 4 %
SOR END EOR

LADDER 111 "SHIFT TOP"
